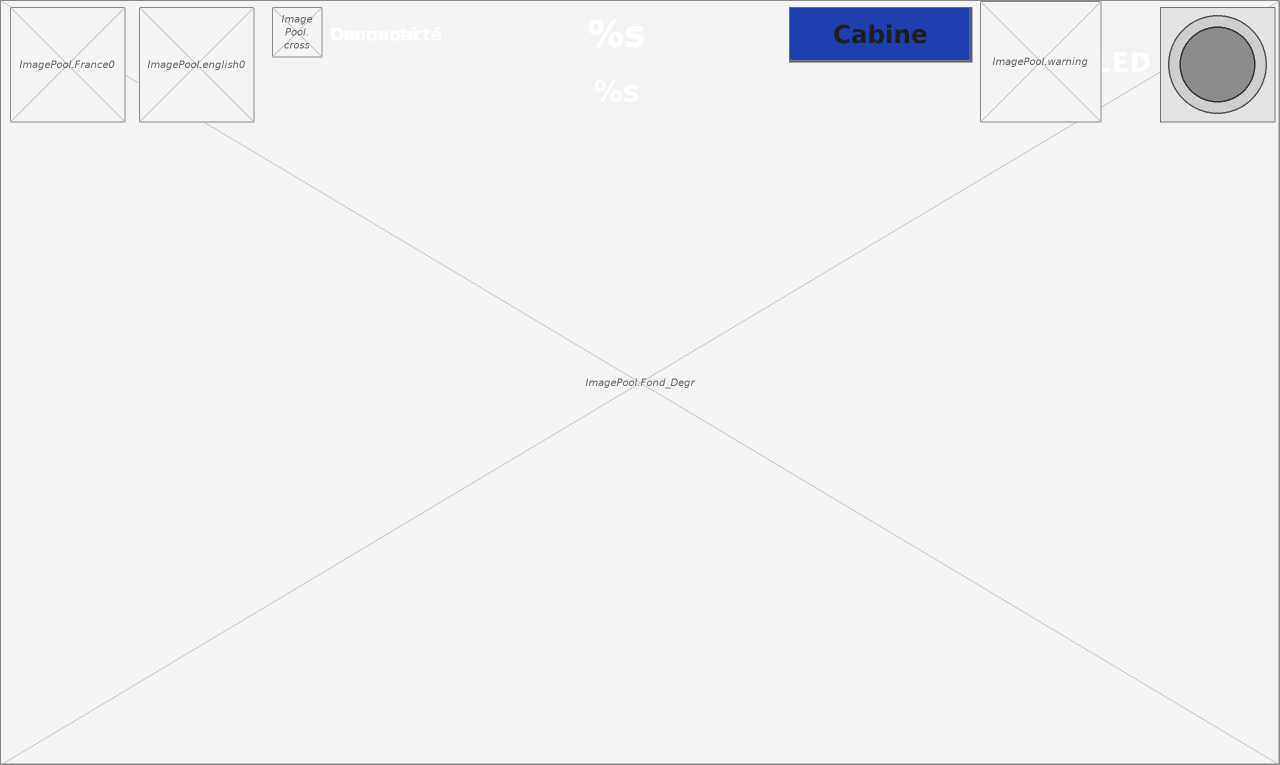
VISUALIZATION masque  // 1280x765
    Image (0,0 1280x765), image: ImagePool.Fond_Degr
    PushSwitch (1160,7 115x115), variable: Activation_Ecl, behaviour: TOGGLE, style: Switch-PushSwitch-Gray
    Image (10,7 115x115), image: ImagePool.France0
        OnMouseDown: ChangeLanguage ChangeLanguage=fr
    Image (139,7 115x115), image: ImagePool.english0
        OnMouseDown: ChangeLanguage ChangeLanguage=En
    Rectangle (262,64 710x55), "%s", text list: 'Etats_Cabine', text index: Sel_Etats_Cabine
        p55702900: GVL_Visu.Couleur_Cabine2
    Rectangle (463,7 309x53), "%s", text variable: GVL_Visu.Nom_Cabine_EN, invisible if: VisuElems.CURRENTLANGUAGE = 'fr'
    Group (272,7 196x53)
        Image (0,0 50x50), image: ImagePool.checked
        Image (0,0 50x50), invisible if: GVL_Visu.Etat_Connexion, image: ImagePool.cross
        Rectangle (55,0 141x55), "Deconnecté", invisible if: GVL_Visu.Etat_Connexion
        Rectangle (55,0 141x55), "Connecté"
    Rectangle (463,7 307x55), "%s", text variable: GVL_Visu.Nom_Cabine_FR, invisible if: VisuElems.CURRENTLANGUAGE = 'en'
    Rectangle (1073,36 81x53), "LED"
    Button (789,7 183x55), "Cabine"
        OnMouseDown: OpenDialog Dialog=Actionneurs, OpenModal=True, PositionX=0, PositionY=0
    Group (980,1 121x121)
        Image (2,4 113x113), invisible if: GVL_Visu.On_Off_Anim_Lent OR NOT Mode_Warning, image: ImagePool.caution
            OnMouseDown: OpenDialog Dialog=Alarmes, OpenModal=True, PositionX=0, PositionY=0
        Image (0,0 121x121), invisible if: GVL_Visu.On_Off_Anim_Lent OR NOT Mode_Cabine_Defaut, image: ImagePool.warning
            OnMouseDown: OpenDialog Dialog=Alarmes, OpenModal=True, PositionX=0, PositionY=0
END_VISUALIZATION

(* stored: Version 1.1.0.1, ProductVersion 3.1.4024.15
   Visu masque: Id {e9e40cab-8594-4572-a903-7a06237479b2} *)
